// TIA Portal V21 export
VAR_GLOBAL   // PLC tag table "K_NumSistema"
END_VAR
VAR_GLOBAL CONSTANT   // user constants
   K_NumKTipo : Int := 16;   // Numero di KTipo presenti nel programma
   K_NumPercorso : Int := 0;
   K_NumUtente : Int := 0;
   K_NumPopup : Int := 1;
   K_NumCamma : Int := 0;
   K_NumValvolaFestoVTEM : Int := 0;
   K_NumVistaManuale : Int := 0;
   K_NumSezionePastorizzatore : Int := 0;
   K_NumSegnaleMacchina : Int := 2;   // Numero di macchine con cui abbiamo segnali
   K_NumSegnaleMacchinaDigitale : Int := 6;
   K_NumSegnaleMacchinaAnalogico : Int := 0;
   K_NumConteggio : Int := 0;
   K_NumFrontiSalitaDiscesa : Int := 0;
   K_NumRifIncrociatiSequenza : Int := 5;   // Rappresenta il numero di riferimenti incrociti possibili delle sequenze (Una valvola può essere comandata da più sequenze)
   K_NumPassi : Int := 25;   // Numero di passi per ogni sequenza
   K_NumDatiBool_Ricetta : Int := 10;
   K_NumDatiReal_Ricetta : Int := 10;
   K_NumTrends : Int := 0;
END_VAR
